// TIA Portal V21 export
// export: Created 2026-07-04T05:03:44.7534001Z, ExportSetting None, DisplayName Totally Integrated Automation Portal, DisplayVersion V21, DisplayName SINAMICS Startdrive Advanced, DisplayVersion V21, DisplayName SINAMICS Startdrive G110M, G120, G120C, G120D, G120P, G115D, DisplayVersion V21, DisplayName SINAMICS Startdrive G130, G150, S120, S150, G200, G220, S200, S210, S220, Innomotics MVD, DisplayVersion V21, DisplayName STEP 7 Professional, DisplayVersion V21, DisplayName STEP 7 Safety, DisplayVersion V21, DisplayName Tech WebApplication, DisplayVersion V21, DisplayName WinCC Basic/Comfort/Advanced, DisplayVersion V21, DisplayName WinCC Professional, DisplayVersion V21, DisplayName WinCC Unified, DisplayVersion V21
FUNCTION_BLOCK "FlowControl_SCL"   // FB2101, LAD
{ S7_Optimized_Access := 'TRUE' }
// stored: AutoNumber false, MemoryReserve 100, SetENOAutomatically false
   VAR_INPUT
      启用 : Bool;   // 使能流程控制FB，FALSE时不允许启动
      启动 : Bool;   // 启动命令，条件满足时进入步骤1
      停止 : Bool;   // 正常停止命令，停止运行并把当前步清零
      暂停 : Bool;   // 暂停命令，保持当前步不继续推进
      复位 : Bool;   // 复位命令，清除完成/故障/暂停并把当前步清零
      中止 : Bool;   // 中止命令，强制退出流程并把当前步清零
      启动允许 : Bool;   // 启动允许条件，例如安全、气压、伺服Ready等
      联锁正常 : Bool;   // 运行中联锁正常，FALSE时触发故障
   END_VAR
   VAR_OUTPUT
      就绪 : Bool;   // 可启动状态：启用、允许、无运行、无故障、未完成
      运行中 : Bool;   // 流程运行锁存状态
      完成 : Bool;   // 流程正常完成，需要复位清除
      故障 : Bool;   // 流程异常停止，需要复位清除
      已暂停 : Bool;   // 流程暂停锁存状态
      当前步 : Int;   // 当前流程步骤号，流程段直接MOVE维护
      故障代码 : Word;   // 故障代码，257表示运行中联锁断开
   END_VAR
   VAR
      启动边沿 : Bool;   // SCL条件段中记录启动命令上一扫描周期状态
      完成边沿 : Bool;   // 完成P上升沿线圈的边沿存储位
      IEC_Timer_0_Instance : TON_TIME;
      IEC_Timer_0_Instance_1 : TON_TIME;
   END_VAR
   VAR_TEMP   // added for the SCL form of the ladder/FBD networks
      _w1 : Bool;
   END_VAR
BEGIN

REGION Network 1 (SCL): 条件判断集中处理
   // 复位、启动、暂停、联锁、停止和就绪输出集中放在本SCL程序段；流程步骤仍在后续梯形图段维护。
   // 复位/中止：最高优先级，清除全部流程状态
   IF #复位 OR #中止 THEN
       #运行中 := FALSE;
       #已暂停 := FALSE;
       #完成 := FALSE;
       #故障 := FALSE;
       #当前步 := 0;
       #故障代码 := W#16#0000;

   // 停止：正常退出流程，只停止运行并回到0步
   ELSIF #停止 THEN
       #运行中 := FALSE;
       #已暂停 := FALSE;
       #当前步 := 0;

   ELSE
       // 暂停保持：运行中收到暂停命令后锁存暂停状态
       IF #运行中 AND #暂停 THEN
           #已暂停 := TRUE;
       END_IF;

       // 暂停恢复：运行中暂停命令撤销后清除暂停状态
       IF #运行中 AND NOT #暂停 THEN
           #已暂停 := FALSE;
       END_IF;

       // 联锁保护：运行中联锁断开时报警并停止运行
       IF #运行中 AND NOT #联锁正常 THEN
           #故障 := TRUE;
           #运行中 := FALSE;
           #故障代码 := W#16#0101; // 十进制257
       END_IF;

       // 启动条件：启动命令上升沿且所有条件满足时进入步骤1
       IF #启用
          AND #启动 AND NOT #启动边沿
          AND #启动允许
          AND #联锁正常
          AND NOT #运行中
          AND NOT #故障
          AND NOT #复位
          AND NOT #中止
          AND NOT #停止 THEN
           #运行中 := TRUE;
           #完成 := FALSE;
           #当前步 := 1;
       END_IF;
   END_IF;

   // 就绪输出：外部可以用它判断当前是否允许重新给启动上升沿
   #就绪 := #启用
          AND NOT #启动
          AND #启动允许
          AND #联锁正常
          AND NOT #运行中
          AND NOT #故障
          AND NOT #中止;

   // 启动边沿存储：放在条件段最后，供下一扫描周期判断上升沿
   #启动边沿 := #启动;
END_REGION

REGION Network 2: 步骤1程序段
   // 当前步等于1且未暂停时，TON计时5秒，计时完成后MOVE 2进入下一步。
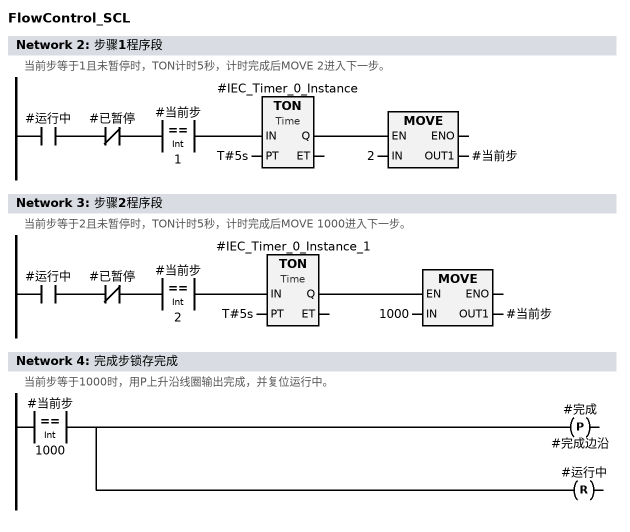
   RUNG wire#powerrail
      Contact( #运行中 )
      I_Contact( #已暂停 )
      { S7_Templates := "SrcType := Int" } EQ_Contact(in1 := #当前步, in2 := 1)
      { S7_Templates := "time_type := Time" } #IEC_Timer_0_Instance.TON(pt := T#5s, et =>)
      { S7_GenerateENO := "TRUE" } Move(in := 2, out1 => #当前步)
   END_RUNG
   // the same network as SCL:
   #IEC_Timer_0_Instance(IN := #运行中 AND NOT #已暂停 AND (#当前步 = 1), PT := T#5s);   // TON
   IF #IEC_Timer_0_Instance.Q THEN #当前步 := 2; END_IF;
END_REGION

REGION Network 3: 步骤2程序段
   // 当前步等于2且未暂停时，TON计时5秒，计时完成后MOVE 1000进入下一步。
   RUNG wire#powerrail
      Contact( #运行中 )
      I_Contact( #已暂停 )
      { S7_Templates := "SrcType := Int" } EQ_Contact(in1 := #当前步, in2 := 2)
      { S7_Templates := "time_type := Time" } #IEC_Timer_0_Instance_1.TON(pt := T#5s, et =>)
      { S7_GenerateENO := "TRUE" } Move(in := 1000, out1 => #当前步)
   END_RUNG
   // the same network as SCL:
   #IEC_Timer_0_Instance_1(IN := #运行中 AND NOT #已暂停 AND (#当前步 = 2), PT := T#5s);   // TON
   IF #IEC_Timer_0_Instance_1.Q THEN #当前步 := 1000; END_IF;
END_REGION

REGION Network 4: 完成步锁存完成
   // 当前步等于1000时，用P上升沿线圈输出完成，并复位运行中。
   #_w1 := #当前步 = 1000;
   #完成 := #_w1 AND NOT #完成边沿;   // rising edge
   #完成边沿 := #_w1;
   IF #_w1 THEN #运行中 := FALSE; END_IF;
END_REGION
END_FUNCTION_BLOCK
